TYPE ST105_Fanuc_command_t :
STRUCT
    FG_Pick     : BIT; // Pick pieces at the feeder side
    FG_Place    : BIT; // Place pieces at the mover side
    reserve_b2  : BIT; // 
    reserve_b3  : BIT; // 
    reserve_b4  : BIT; // 
    reserve_b5  : BIT; // 
    reserve_b6  : BIT; // 
    reserve_b7  : BIT; // 
    ZOff        : BIT; // negative flag for the Z offset
    XOff        : BIT; // negative flag for the X offset
    YOff        : BIT; // negative flag for the Y offset
    reserve_b11 : BIT; // 
    reserve_b12 : BIT; // 
    reserve_b13 : BIT; // 
    reserve_b14 : BIT; // 
    reserve_b15 : BIT; // 
END_STRUCT
END_TYPE

(* stored: Version 1.1.0.1, ProductVersion 3.1.4024.6
   DUT ST105_Fanuc_command_t: Id {e5ae7b81-47d3-439d-a560-25e2bcd986ca} *)
